// TIA Portal V17 export
// export: Created 2023-02-14T02:49:55.4297619Z, ExportSetting WithDefaults, DisplayName Totally Integrated Automation Portal, DisplayVersion V17, DisplayName TIA Portal Openness, DisplayVersion V17, DisplayName TIA Portal Teamcenter Gateway, DisplayVersion V17, DisplayName TIA Portal Version Control Interface, DisplayVersion V17, DisplayName SINAMICS Startdrive Advanced, DisplayVersion V17, DisplayName SINAMICS Startdrive G130, G150, S120, S150, SINAMICS MV, S210, DisplayVersion V17, DisplayName SINAMICS Startdrive G110M, G120, G120C, G120D, G120P, G115D, DisplayVersion V17, DisplayName STEP 7 Professional, DisplayVersion V17, DisplayName STEP 7 Safety, DisplayVersion V17, DisplayName WinCC Professional, DisplayVersion V17
VAR_GLOBAL   // PLC tag table "MCC Panel Blending"
   "P-13.02 Overload" AT %I0.0 : Bool;   // CIP RETURN PUMP HOMOMIXER AREA
   "P-22.02 Overload" AT %I0.1 : Bool;   // BYPASS CIP PUMP REWORK TANK T-22.00
   "P-32.02 Overload" AT %I0.2 : Bool;   // BYPASS CIP PUMP REWORK TANK T-32.00
   "P-13.02 Feedback" AT %I0.3 : Bool;   // CIP RETURN PUMP HOMOMIXER AREA
   "P-22.02 Feedback" AT %I0.4 : Bool;   // BYPASS CIP PUMP REWORK TANK T-22.00
   "P-32.02 Feedback" AT %I0.5 : Bool;   // BYPASS CIP PUMP REWORK TANK T-32.00
   "Emergency Stop MCC Panel Blending" AT %I0.6 : Bool;   // Emergency Stop MCC Panel Blending
   "P-34.02 Overload" AT %I0.7 : Bool;   // CIP RETURN PUMP STORAGE AREA TO CIP RETURN LINE 3
   "P-34.02 Feedback" AT %I1.0 : Bool;   // CIP RETURN PUMP STORAGE AREA TO CIP RETURN LINE 3
   "P-34.01 Feedback" AT %I1.1 : Bool;
   "XA-14.01 Alarm" AT %I1.2 : Bool;
   "XA-14.01 Feedback" AT %I1.3 : Bool;
   "P-81.02 Overload" AT %I1.4 : Bool;
   "P-81.02 Feedback" AT %I1.5 : Bool;
   "P-81.01 Feedback" AT %I1.6 : Bool;
   "P-82.01 Alarm" AT %I1.7 : Bool;
   "P-82.01 Feedback" AT %I2.0 : Bool;
   "P-84.01 Alarm" AT %I2.1 : Bool;
   "P-84.01 Feedback" AT %I2.2 : Bool;
   "P-84.02 Alarm" AT %I2.3 : Bool;
   "P-84.02 Feedback" AT %I2.4 : Bool;
   "P-24.02 Overload" AT %I2.5 : Bool;
   "P-24.02 Feedback" AT %I2.6 : Bool;
   "P-82.02 Overload" AT %I2.7 : Bool;
   "P-82.02 Feedback" AT %I3.0 : Bool;
   "P-84-03 Overload" AT %I3.1 : Bool;
   "P-84.03 Feedback" AT %I3.2 : Bool;
   "P-84.04 Overload" AT %I3.3 : Bool;
   "P-84.04 Feedback" AT %I3.4 : Bool;
   "MCC spare 21" AT %I3.5 : Bool;
   "MCC spare 22" AT %I3.6 : Bool;
   "MCC spare 23" AT %I3.7 : Bool;
   "XA-12.01 SW" AT %IW700 : Word;
   "XA-12.01 AV" AT %IW702 : Int;
   "XA-12.01 Voltage" AT %IW704 : Int;
   "XA-12.01 Ampere" AT %IW706 : Int;
   "XA-12.01 KW" AT %IW708 : Int;
   "XA-12.01 Nm" AT %IW710 : Int;
   "XA-13.01 SW" AT %IW712 : Word;
   "XA-13.01 AV" AT %IW714 : Int;
   "XA-13.01 Voltage" AT %IW716 : Int;
   "XA-13.01 Ampere" AT %IW718 : Int;
   "XA-13.01 KW" AT %IW720 : Int;
   "XA-13.01 Nm" AT %IW722 : Int;
   "XA-20.00 SW" AT %IW724 : Word;
   "XA-20.00 AV" AT %IW726 : Int;
   "XA-20.00 Voltage" AT %IW728 : Int;
   "XA-20.00 Ampere" AT %IW730 : Int;
   "XA-20.00 KW" AT %IW732 : Int;
   "XA-20.00 Nm" AT %IW734 : Int;
   "XA-21.00 SW" AT %IW736 : Word;
   "XA-21.00 AV" AT %IW738 : Int;
   "XA-21.00 Voltage" AT %IW740 : Int;
   "XA-21.00 Ampere" AT %IW742 : Int;
   "XA-21.00 KW" AT %IW744 : Int;
   "XA-21.00 Nm" AT %IW746 : Int;
   "P-21.01 SW" AT %IW748 : Word;
   "P-21.01 AV" AT %IW750 : Int;
   "P-21.01 Voltage" AT %IW752 : Int;
   "P-21.01 Ampere" AT %IW754 : Int;
   "P-21.01 KW" AT %IW756 : Int;
   "P-21.01 Nm" AT %IW758 : Int;
   "P-22.01 SW" AT %IW760 : Word;
   "P-22.01 AV" AT %IW762 : Int;
   "P-22.01 Voltage" AT %IW764 : Int;
   "P-22.01 Ampere" AT %IW766 : Int;
   "P-22.01 KW" AT %IW768 : Int;
   "P-22.01 Nm" AT %IW770 : Int;
   "P-22.03 SW" AT %IW772 : Word;
   "P-22.03 AV" AT %IW774 : Int;
   "P-22.03 Voltage" AT %IW776 : Int;
   "P-22.03 Ampere" AT %IW778 : Int;
   "P-22.03 KW" AT %IW780 : Int;
   "P-22.03 Nm" AT %IW782 : Int;
   "P-23.01 SW" AT %IW784 : Word;
   "P-23.01 AV" AT %IW786 : Int;
   "P-23.01 Voltage" AT %IW788 : Int;
   "P-23.01 Ampere" AT %IW790 : Int;
   "P-23.01 KW" AT %IW792 : Int;
   "P-23.01 Nm" AT %IW794 : Int;
   "P-24.01 SW" AT %IW796 : Word;
   "P-24.01 AV" AT %IW798 : Int;
   "P-24.01 Voltage" AT %IW800 : Int;
   "P-24.01 Ampere" AT %IW802 : Int;
   "P-24.01 KW" AT %IW804 : Int;
   "P-24.01 Nm" AT %IW806 : Int;
   "XA-30.00 SW" AT %IW820 : Word;
   "XA-30.00 AV" AT %IW822 : Int;
   "XA-30.00 Voltage" AT %IW824 : Int;
   "XA-30.00 Ampere" AT %IW826 : Int;
   "XA-30.00 KW" AT %IW828 : Int;
   "XA-30.00 Nm" AT %IW830 : Int;
   "XA-31.00 SW" AT %IW832 : Word;
   "XA-31.00 AV" AT %IW834 : Int;
   "XA-31.00 Voltage" AT %IW836 : Int;
   "XA-31.00 Ampere" AT %IW838 : Int;
   "XA-31.00 KW" AT %IW840 : Int;
   "XA-31.00 Nm" AT %IW842 : Int;
   "P-31.01 SW" AT %IW844 : Word;
   "P-31.01 AV" AT %IW846 : Int;
   "P-31.01 Voltage" AT %IW848 : Int;
   "P-31.01 Ampere" AT %IW850 : Int;
   "P-31.01 KW" AT %IW852 : Int;
   "P-31.01 Nm" AT %IW854 : Int;
   "P-32.01 SW" AT %IW856 : Word;
   "P-32.01 AV" AT %IW858 : Int;
   "P-32.01 Voltage" AT %IW860 : Int;
   "P-32.01 Ampere" AT %IW862 : Int;
   "P-32.01 KW" AT %IW864 : Int;
   "P-32.01 Nm" AT %IW866 : Int;
   "P-32.03 SW" AT %IW868 : Word;
   "P-32.03 AV" AT %IW870 : Int;
   "P-32.03 Voltage" AT %IW872 : Int;
   "P-32.03 Ampere" AT %IW874 : Int;
   "P-32.03 KW" AT %IW876 : Int;
   "P-32.03 Nm" AT %IW878 : Int;
   "P-35.01 SW" AT %IW880 : Word;
   "P-35.01 AV" AT %IW882 : Int;
   "P-35.01 Voltage" AT %IW884 : Int;
   "P-35.01 Ampere" AT %IW886 : Int;
   "P-35.01 KW" AT %IW888 : Int;
   "P-35.01 Nm" AT %IW890 : Int;
   "P-34.01 Act Speed" AT %IW684 : Int;
   "XA-14.01 Act Speed" AT %IW686 : Int;
   "P-81.01 Act Speed" AT %IW696 : Int;
   "P-82.01 Act Speed" AT %IW690 : Int;
   "P-84.01 Act Speed" AT %IW692 : Int;
   "P-84.02 Act Speed" AT %IW694 : Int;
   "P-34.01 SW" AT %IW808 : Word;
   "P-34.01 AV" AT %IW810 : Int;
   "P-34.01 Voltage" AT %IW812 : Int;
   "P-34.01 Ampere" AT %IW814 : Int;
   "P-34.01 KW" AT %IW816 : Int;
   "P-34.01 Nm" AT %IW818 : Int;
   "P-20.01 SW" AT %IW972 : Int;
   "P-20.01 AV" AT %IW974 : Int;
   "P-20.01 Voltage" AT %IW976 : Int;
   "P-20.01 Ampere" AT %IW978 : Int;
   "P-20.01 KW" AT %IW980 : Int;
   "P-20.01 Nm" AT %IW982 : Int;
   "P-30.01 SW" AT %IW1080 : Int;
   "P-30.01 AV" AT %IW1082 : Int;
   "P-30.01 Voltage" AT %IW1084 : Int;
   "P-30.01 Ampere" AT %IW1086 : Int;
   "P-30.01 KW" AT %IW1088 : Int;
   "P-30.01 Nm" AT %IW1090 : Int;
   "P-40.01 SW" AT %IW1092 : Int;
   "P-40.01 AV" AT %IW1094 : Int;
   "P-40.01 Voltage" AT %IW1096 : Int;
   "P-40.01 Ampere" AT %IW1098 : Int;
   "P-40.01 KW" AT %IW1100 : Int;
   "P-40.01 Nm" AT %IW1102 : Int;
   "P-41.01 SW" AT %IW1104 : Int;
   "P-41.01 AV" AT %IW1106 : Int;
   "P-41.01 Voltage" AT %IW1108 : Int;
   "P-41.01 Ampere" AT %IW1110 : Int;
   "P-41.01 KW" AT %IW1112 : Int;
   "P-41.01 Nm" AT %IW1114 : Int;
   "XA-40.00 SW" AT %IW1116 : Int;
   "XA-40.00 AV" AT %IW1118 : Int;
   "XA-40.00 Voltage" AT %IW1120 : Int;
   "XA-40.00 Ampere" AT %IW1122 : Int;
   "XA-40.00 KW" AT %IW1124 : Int;
   "XA-40.00 Nm" AT %IW1126 : Int;
   "XA-41.00 SW" AT %IW1128 : Int;
   "XA-41.00 AV" AT %IW1130 : Int;
   "XA-41.00 Voltage" AT %IW1132 : Int;
   "XA-41.00 Ampere" AT %IW1134 : Int;
   "XA-41.00 KW" AT %IW1136 : Int;
   "XA-41.00 Nm" AT %IW1138 : Int;
   "P-13.02 OUT" AT %Q0.0 : Bool;   // CIP RETURN PUMP HOMOMIXER AREA
   "P-81.02 OUT" AT %Q0.1 : Bool;
   "P-22.04 OUT" AT %Q0.2 : Bool;
   "P-34.02 OUT" AT %Q0.3 : Bool;
   "P-32.04 OUT" AT %Q0.4 : Bool;
   "P-81.01 OUT" AT %Q0.5 : Bool;
   "P-34.01 OUT" AT %Q0.6 : Bool;
   "XA-14.01 OUT" AT %Q0.7 : Bool;
   "P-82.01 OUT" AT %Q1.0 : Bool;
   "P-84.01 OUT" AT %Q1.1 : Bool;
   "P-84.02 OUT" AT %Q1.2 : Bool;
   "P-24.02 OUT" AT %Q1.3 : Bool;
   "P-82.02 OUT" AT %Q1.4 : Bool;
   "P-84.03 OUT" AT %Q1.5 : Bool;
   "P-84.04 OUT" AT %Q1.6 : Bool;
   "MCC spare 35" AT %Q1.7 : Bool;
   "XA-12.01 CW" AT %QW700 : Word;
   "XA-12.01 SP" AT %QW702 : Word;
   "XA-13.01 CW" AT %QW712 : Word;
   "XA-13.01 SP" AT %QW714 : Word;
   "XA-20.00 CW" AT %QW724 : Word;
   "XA-20.00 SP" AT %QW726 : Word;
   "XA-21.00 CW" AT %QW736 : Word;
   "XA-21.00 SP" AT %QW738 : Word;
   "P-21.01 CW" AT %QW748 : Word;
   "P-21.01 SP" AT %QW750 : Word;
   "P-22.01 CW" AT %QW760 : Word;
   "P-22.01 SP" AT %QW762 : Word;
   "P-22.03 CW" AT %QW772 : Word;
   "P-22.03 SP" AT %QW774 : Word;
   "P-23.01 CW" AT %QW784 : Word;
   "P-23.01 SP" AT %QW786 : Word;
   "P-24.01 CW" AT %QW796 : Word;
   "P-24.01 SP" AT %QW798 : Word;
   "XA-30.00 CW" AT %QW820 : Word;
   "XA-30.00 SP" AT %QW822 : Word;
   "XA-31.00 CW" AT %QW832 : Word;
   "XA-31.00 SP" AT %QW834 : Word;
   "P-31.01 CW" AT %QW844 : Word;
   "P-31.01 SP" AT %QW846 : Word;
   "P-32.01 CW" AT %QW856 : Word;
   "P-32.01 SP" AT %QW858 : Word;
   "P-32.03 CW" AT %QW868 : Word;
   "P-32.03 SP" AT %QW870 : Word;
   "P-35.01 CW" AT %QW880 : Word;
   "P-35.01 SP" AT %QW882 : Word;
   "P-34.01 SP Speed" AT %QW98 : Int;
   "XA-14.01 SP Speed" AT %QW100 : Int;
   "P-81.01 SP Speed" AT %QW102 : Int;
   "P-82.01 SP Speed" AT %QW104 : Int;
   "P-84.01 SP Speed" AT %QW106 : Int;
   "P-84.02 SP Speed" AT %QW108 : Int;
   "P-34.01 CW" AT %QW808 : Word;
   "P-34.01 SP" AT %QW810 : Word;
   "P-20.01 CW" AT %QW972 : Int;
   "P-20.01 SP" AT %QW974 : Int;
   "P-30.01 CW" AT %QW1080 : Int;
   "P-30.01 SP" AT %QW1082 : Int;
   "P-40.01 CW" AT %QW1092 : Int;
   "P-40.01 SP" AT %QW1094 : Int;
   "P-41.01 CW" AT %QW1104 : Int;
   "P-41.01 SP" AT %QW1106 : Int;
   "XA-40.00 CW" AT %QW1116 : Int;
   "XA-40.00 SP" AT %QW1118 : Int;
   "XA-41.00 CW" AT %QW1128 : Int;
   "XA-41.00 SP" AT %QW1130 : Int;
END_VAR
